FUNCTION_BLOCK FB_Component_ServoMotor IMPLEMENTS I_Component
VAR_INPUT
	bEnable				: BOOL;	

	bHomingSensor		: BOOL;
	bHomingSpeed		: INT;
	uMaxRPM				: INT;
	bSetCounterDone		: BOOL;
	rGearRatio			: REAL;
END_VAR
VAR_IN_OUT
	
	bSetCounter			: BOOL;
	dSetCounterValue	: DINT;
	bEnableDrive		: BOOL;
	uAnalogOut			: INT;
END_VAR
VAR_OUTPUT
	uCurrRPM			: INT;
END_VAR
VAR
	tHomeTrig			: F_TRIG;
	bHomeTriggered		: BOOL;
END_VAR

(*

aOutServo2						AT %Q*	: INT;	// term 18.1

bSetCounterDoneServo2			AT %I*	: BOOL;
dCountServo2					AT %I*	: DINT;

dSetCounterServo2				AT %Q*	: BOOL;
dSetCounterValueServo2			AT %Q*	: DINT;
*)

IF bEnable THEN
	uCurrRPM := REAL_TO_INT((((INT_TO_REAL(ABS(uAnalogOut))/32767)) * uMaxRPM) / rGearRatio);
ELSE
	bEnableDrive := FALSE;
	uAnalogOut	 := 0;
	uCurrRPM	 := 0;
END_IF

{warning 'add method implementation '}
METHOD M_Halt : BOOL
END_METHOD

{warning 'add method implementation '}
METHOD M_Start : BOOL
END_METHOD

{warning 'add method implementation '}
METHOD M_Stop : BOOL
END_METHOD

END_FUNCTION_BLOCK

(* stored: Version 1.1.0.1, ProductVersion 3.1.4024.15
   POU FB_Component_ServoMotor: Id {7bc5585d-e043-4a4d-90c5-3748dca72298}, SpecialFunc None
   Method M_Halt: Id {e670ceb9-7bbb-4f32-865f-4279a3ed37e2}
   Method M_Start: Id {5850c2fb-1fd2-46fc-baa0-6de215783738}
   Method M_Stop: Id {a7e4a841-9d33-4e88-80db-37d91db85604} *)
